Universal Robots PolyScope program: xiaomi.urp

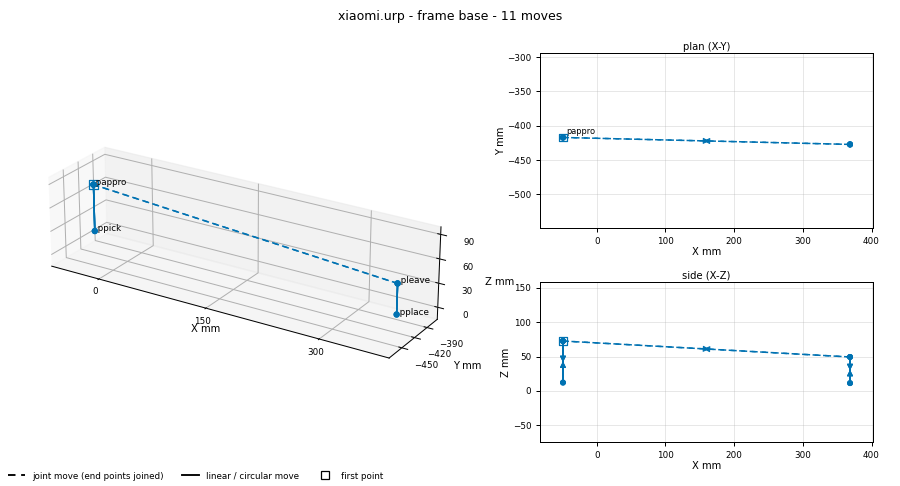
[picture p0: tool path of xiaomi.urp in frame base, 11 of 11 moves have a stored position in this frame; points joined in program order, loops and branches not executed]
Program xiaomi (installation=20240827 directory=/programs/Demos/adaptiveGrip createdIn=5.15.1 lastSavedIn=5.15.1 robotSerialNumber=20245500285)
Calibrated DH parameters: a=[0.000097, -0.210459, -0.026602, 0.000137, 0.000078, 0]; d=[0.162601, 254.180657, -54.076236, -199.970743, 0.099615, 0.099684]; alpha=[1.569796, -0.001455, 0.001957, 1.570525, -1.571561, 0]; deltaTheta=[0, -1.053331, 8.839472, -1.50296, 0.000002, 0]
InitVariablesNode
BeforeStart
  SuppressedNode
    MoveL speed 250 mm/s, acceleration 1200 mm/s^2 (useActiveTCP=true) feature=Base
      Waypoint ppick: TCP in base x=-36.634 y=-638.502 z=14.663 mm, rx=2.1795 ry=2.2626 rz=-0.0001 rad; joints [74.558, -61.012, 96.454, -125.49, -90.074, 72.599] deg; TCP offset x=-0.17 y=0 z=192.95 mm, rx=0 ry=0 rz=0 rad
      Waypoint pappro: TCP in base x=-36.657 y=-638.51 z=49.536 mm, rx=2.1795 ry=2.2625 rz=-0.0002 rad; joints [74.558, -63.595, 94.504, -120.959, -90.063, 72.602] deg
  Script: usb = rpc_factory("xmlrpc","http://192.168.1.7:9120/RPC2")
  Script: usb.open()
Robot Program (runOnlyOnce=false)
  MoveJ speed 180 deg/s, acceleration 720 deg/s^2 (useActiveTCP=true) feature=Base
    Waypoint pappro: motionParameters(blendRadius=0.01); TCP in base x=-49.281 y=-417.157 z=72.654 mm, rx=2.1934 ry=2.2491 rz=-0.0002 rad; joints [64.617, -93.36, 127.824, -124.513, -90.042, 63.331] deg
  Script: usb.open()
  MoveL speed 1000 mm/s, acceleration 2000 mm/s^2 (useActiveTCP=true) feature=Base
    Waypoint ppick: TCP in base x=-49.302 y=-417.173 z=12.122 mm, rx=2.1935 ry=2.2491 rz=-0.0003 rad; joints [64.616, -86.456, 132.517, -136.116, -90.066, 63.326] deg
  Script: usb.adaptiveClose()
  MoveL speed 1000 mm/s, acceleration 2000 mm/s^2 (useActiveTCP=true) feature=Base
    Waypoint pappro: TCP in base x=-49.281 y=-417.157 z=72.654 mm, rx=2.1934 ry=2.2491 rz=-0.0002 rad; joints [64.617, -93.36, 127.824, -124.513, -90.042, 63.331] deg
  MoveJ speed 180 deg/s, acceleration 720 deg/s^2 (useActiveTCP=true) feature=Base
    Waypoint pleave: motionParameters(blendRadius=0.03); TCP in base x=368.713 y=-427.279 z=49.429 mm, rx=-2.1647 ry=-2.2768 rz=0.0001 rad; joints [117.016, -72.462, 107.675, -125.258, -90.064, 114.298] deg
  MoveL speed 1000 mm/s, acceleration 2000 mm/s^2 (useActiveTCP=true) feature=Base
    Waypoint pplace: TCP in base x=368.741 y=-427.273 z=11.348 mm, rx=2.1646 ry=2.2768 rz=-0.0001 rad; joints [117.017, -69.125, 109.891, -130.812, -90.076, 114.292] deg
  Script: usb.open()
  MoveL speed 1000 mm/s, acceleration 2000 mm/s^2 (useActiveTCP=true) feature=Base
    Waypoint pleave: TCP in base x=368.713 y=-427.279 z=49.429 mm, rx=-2.1647 ry=-2.2768 rz=0.0001 rad; joints [117.016, -72.462, 107.675, -125.258, -90.064, 114.298] deg
  MoveL speed 1000 mm/s, acceleration 2000 mm/s^2 (useActiveTCP=true) feature=Base
    Waypoint pplace: TCP in base x=368.741 y=-427.273 z=11.348 mm, rx=2.1646 ry=2.2768 rz=-0.0001 rad; joints [117.017, -69.125, 109.891, -130.812, -90.076, 114.292] deg
    Script: usb.adaptiveClose()
  MoveL speed 1000 mm/s, acceleration 2000 mm/s^2 (useActiveTCP=true) feature=Base
    Waypoint pleave: TCP in base x=368.713 y=-427.279 z=49.429 mm, rx=-2.1647 ry=-2.2768 rz=0.0001 rad; joints [117.016, -72.462, 107.675, -125.258, -90.064, 114.298] deg
  MoveJ speed 180 deg/s, acceleration 360 deg/s^2 (useActiveTCP=true) feature=Base
    Waypoint pappro: TCP in base x=-49.281 y=-417.157 z=72.654 mm, rx=2.1934 ry=2.2491 rz=-0.0002 rad; joints [64.617, -93.36, 127.824, -124.513, -90.042, 63.331] deg
  MoveL speed 1000 mm/s, acceleration 6000 mm/s^2 (useActiveTCP=true) feature=Base
    Waypoint ppick: TCP in base x=-49.302 y=-417.173 z=12.122 mm, rx=2.1935 ry=2.2491 rz=-0.0003 rad; joints [64.616, -86.456, 132.517, -136.116, -90.066, 63.326] deg
    Script: usb.open()
  MoveL speed 1000 mm/s, acceleration 6000 mm/s^2 (useActiveTCP=true) feature=Base
    Waypoint pappro: TCP in base x=-49.281 y=-417.157 z=72.654 mm, rx=2.1934 ry=2.2491 rz=-0.0002 rad; joints [64.617, -93.36, 127.824, -124.513, -90.042, 63.331] deg
